// TwinCAT 3 PLC project Main
// ProgramVersion: 3.1.4023.0
// libraries:
//   Tc2_Standard, * (Beckhoff Automation GmbH)
//   Tc2_System, * (Beckhoff Automation GmbH)
//   Tc2_Utilities, * (Beckhoff Automation GmbH)
//   Tc3_Module, * (Beckhoff Automation GmbH)
// project tree:
//   DUTs/ E_EventType.TcDUT, ST_Event.TcDUT
//   / PlcTask.TcTTO
//   POUs/ EventLogger.TcPOU, MAIN.TcPOU, UpdateEventTimeStampWithSystemTime.TcPOU
// real-time tasks:
//   TASK PlcTask: cycle T#10ms, priority 6, ADS port 350

CONFIGURATION Main
    RESOURCE PLC ON TwinCAT3
        TASK PlcTask(INTERVAL := T#10ms, PRIORITY := 6);
        PROGRAM MAIN WITH PlcTask : MAIN;
    END_RESOURCE
END_CONFIGURATION

// ---- DUTs/E_EventType.TcDUT
{attribute 'qualified_only'}
{attribute 'strict'}
TYPE E_EventType :
(
	Alarm := 0,
	Message := 1
);
END_TYPE

// ---- DUTs/ST_Event.TcDUT
TYPE ST_Event :
STRUCT
	eEventType : E_EventType;
	eEventSeverity : TcEventSeverity;
	nEventIdentity : UDINT;
	sEventText: STRING(255);
	dtTimestamp: DATE_AND_TIME;
END_STRUCT
END_TYPE

// ---- POUs/MAIN.TcPOU
PROGRAM MAIN
VAR
	//stTestInstance : ST_Event;
	bBoolean : BOOL := FALSE;
	
	eEventType1 : E_EventType := E_EventType.Alarm;
	eEventSeverity1 : TcEventSeverity := TcEventSeverity.Critical;
	nEventIdentity1 : UDINT := 42;
	sEventText1: STRING(255) := 'spooky event';
	
	EventLogger : EventLogger;
END_VAR

(*IF NOT bBoolean THEN
	UpdateEventTimeStampWithSystemTime(stEvent := stTestInstance);
	bBoolean := TRUE;
END_IF *)

IF bBoolean THEN
	EventLogger.AddEvent(eEventType1, eEventSeverity1, nEventIdentity1, sEventText1);
	bBoolean := FALSE;
END_IF

END_PROGRAM

// ---- POUs/EventLogger.TcPOU
FUNCTION_BLOCK EventLogger
VAR
	EventBuffer : ARRAY[1..MAXIMUM_SIZE_OF_EVENT_BUFFER] OF ST_Event;
	CurrentEventBufferIndex : INT := 0;
END_VAR
VAR CONSTANT
	MAXIMUM_SIZE_OF_EVENT_BUFFER : INT := 100;
END_VAR

(*Returns TRUE if add was succesful and FALSE if buffer is full*)
METHOD AddEvent : BOOL
VAR_INPUT
	eEventType : E_EventType;
	eEventSeverity : TcEventSeverity;
	nEventIdentity : UDINT;
	sEventText: STRING(255);
END_VAR
IF IsEventBufferFull() THEN
	CurrentEventBufferIndex := CurrentEventBufferIndex + 1;
	EventBuffer[CurrentEventBufferIndex].eEventType := eEventType;
	EventBuffer[CurrentEventBufferIndex].eEventSeverity := eEventSeverity;
	EventBuffer[CurrentEventBufferIndex].nEventIdentity := nEventIdentity;
	EventBuffer[CurrentEventBufferIndex].sEventText := sEventText;
	UpdateEventTimeStampWithSystemTime(stEvent := EventBuffer[CurrentEventBufferIndex]);
	AddEvent:= TRUE;
ELSE
	AddEvent:= FALSE;
END_IF
END_METHOD

METHOD PRIVATE IsEventBufferFull : BOOL
IF (CurrentEventBufferIndex + 1) > MAXIMUM_SIZE_OF_EVENT_BUFFER THEN
	IsEventBufferFull := TRUE;
ELSE
	IsEventBufferFull := FALSE;
END_IF
END_METHOD

END_FUNCTION_BLOCK

// ---- POUs/UpdateEventTimeStampWithSystemTime.TcPOU
FUNCTION UpdateEventTimeStampWithSystemTime
VAR_INPUT
	stEvent : REFERENCE TO ST_Event;
END_VAR
VAR
	fbGETSYSTEMTIME : GETSYSTEMTIME;
	stFileTime : T_FILETIME;
END_VAR

fbGETSYSTEMTIME(timeLoDW => stFileTime.dwLowDateTime,
				timeHiDW => stFileTime.dwHighDateTime);
				
stEvent.dtTimestamp := FILETIME_TO_DT(filetime := stFileTime);

END_FUNCTION
